# B&R Automation Studio project Ladder
Automation Studio 4.12.2.93

## Configuration Config1

### Hardware
```
X20CP1584 : X20CP1584 v1.10.0.0
  Connector IF2:
    ActivateDevice = 1
  ConfigurationID = Ladder_Config1
  Simulation = 1
  FileDevice1
  FileDeviceName1 = USER
  FileDevicePath1 = USER_PATH
```

## Logical view

### Program Logical/Program

#### Variables.var
```iecst
VAR
	n_cicli_man : INT := 10; (*COSTANTE: numero di cicli che eseguiamo prima di andare in manutenzione*)
	t1s : TIME := T#10s; (*COSTANTE: tempo 1 secondo*)
	tFotocamera : TIME := T#10s; (*COSTANTE: tempo che la fotocamera impiega per leggere i dati*)
	n_kit : INT := 10; (*COSTANTE: valore degli item necessari nel kit*)
	CONVon : BOOL; (*MOTORE: motore per far muovere i pezzi*)
	START : BOOL; (*PULSANTE: avvio del ciclo di lavoro*)
	GO : BOOL; (*PULSANTE: pulsante che ravvia il sistema dopo il bloccaggio alla fotocamera*)
	MR : BOOL; (*PULSANTE: reset della manutenzione*)
	RESET_COUNTER : BOOL; (*PULSANTE: serve per resettare il conteggio dei pezzi buoni*)
	ON : BOOL; (*STATO: identifica che il coclo è attivo*)
	MUOVI : BOOL; (*STATO: identifica lo stato del nastro trasportatore attivo*)
	RISULTATI : BOOL; (*STATO: indichiamo che stiamo conforntando i dati della fotocamera*)
	NON_BUONO : BOOL; (*STATO: quando i pezzi contati sono diversi da n_kit*)
	ATTESA_UTENTE : BOOL; (*STATO: quando si aspetta l'intervento dell'operatore*)
	BUONO : BOOL; (*STATO: quanto i pezzi contati sono pari a n_kit*)
	MAN : BOOL; (*STATO: stato di manutenzione*)
	FOTOCAMERA : BOOL; (*STATO: stato in cui la fotocamera sta leggendo i dati*)
	n_items : INT; (*VARIABILE: numero di oggetti nella vaschetta*)
	n_corrette : INT; (*VARIABILE: numero di volte che la fotocamera ha letto n_kit  oggetti*)
END_VAR
```

#### Cyclic.ld
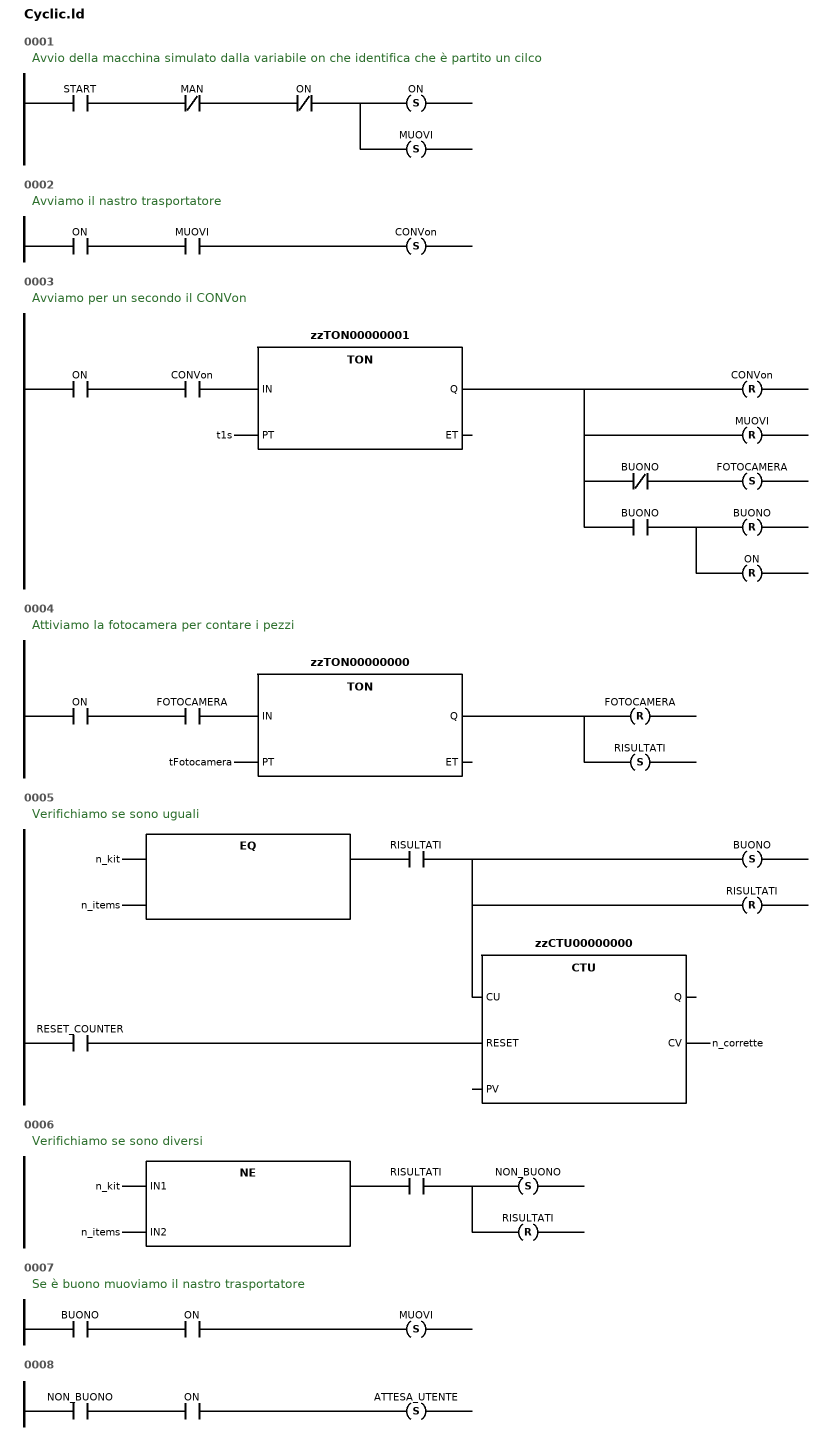
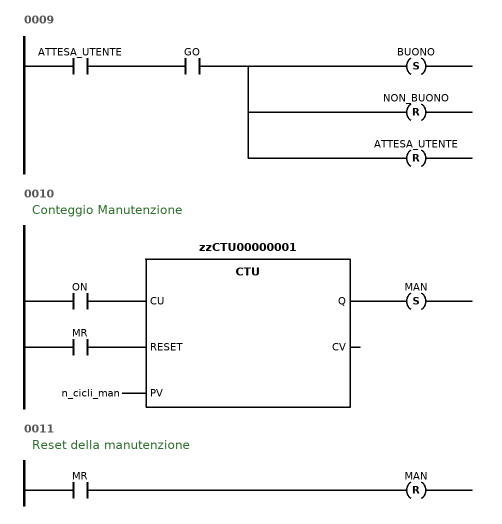
Ladder, written as Structured Text:
```iecst
PROGRAM _CYCLIC
VAR
    _p1 : BOOL;
    _p2 : BOOL;
    _p3 : BOOL;
END_VAR
(* Network 1: Avvio della macchina simulato dalla variabile on che identifica che è partito un cilco *)
_p1 := START AND NOT MAN AND NOT ON;
IF START AND NOT MAN AND NOT ON THEN ON := TRUE; END_IF;
IF _p1 THEN MUOVI := TRUE; END_IF;

(* Network 2: Avviamo il nastro trasportatore *)
IF ON AND MUOVI THEN CONVon := TRUE; END_IF;

(* Network 3: Avviamo per un secondo il CONVon *)
zzTON00000001(IN := ON AND CONVon, PT := t1s);
IF zzTON00000001.Q THEN
    CONVon := FALSE;
    MUOVI := FALSE;
END_IF;
IF zzTON00000001.Q AND NOT BUONO THEN FOTOCAMERA := TRUE; END_IF;
_p2 := zzTON00000001.Q AND BUONO;
IF zzTON00000001.Q AND BUONO THEN BUONO := FALSE; END_IF;
IF _p2 THEN ON := FALSE; END_IF;

(* Network 4: Attiviamo la fotocamera per contare i pezzi *)
zzTON00000000(IN := ON AND FOTOCAMERA, PT := tFotocamera);
IF zzTON00000000.Q THEN
    FOTOCAMERA := FALSE;
    RISULTATI := TRUE;
END_IF;

(* Network 5: Verifichiamo se sono uguali *)
IF (n_kit = n_items) AND RISULTATI THEN BUONO := TRUE; END_IF;
_p3 := (n_kit = n_items) AND RISULTATI;
IF (n_kit = n_items) AND RISULTATI THEN RISULTATI := FALSE; END_IF;
zzCTU00000000(CU := _p3, RESET := RESET_COUNTER);
n_corrette := zzCTU00000000.CV;

(* Network 6: Verifichiamo se sono diversi *)
IF (n_kit <> n_items) AND RISULTATI THEN
    NON_BUONO := TRUE;
    RISULTATI := FALSE;
END_IF;

(* Network 7: Se è buono muoviamo il nastro trasportatore *)
IF BUONO AND ON THEN MUOVI := TRUE; END_IF;

(* Network 8 *)
IF NON_BUONO AND ON THEN ATTESA_UTENTE := TRUE; END_IF;

(* Network 9 *)
IF ATTESA_UTENTE AND GO THEN
    BUONO := TRUE;
    NON_BUONO := FALSE;
    ATTESA_UTENTE := FALSE;
END_IF;

(* Network 10: Conteggio Manutenzione *)
zzCTU00000001(CU := ON, RESET := MR, PV := n_cicli_man);
IF zzCTU00000001.Q THEN MAN := TRUE; END_IF;

(* Network 11: Reset della manutenzione *)
IF MR THEN MAN := FALSE; END_IF;
END_PROGRAM
```
